PROGRAM AnalogConversion
VAR
	i					: INT := 1; //charger 1-6
	j					: INT := 1;  // section 1 - 4 
	k					: INT := 1;  // cap 1-10
	m					: INT := 1; //form cap 1-12
	n					: INT := 6;
	MaxTemp				: INT := 380;
	MinTemp				: INT := -70;
	
	MaxCurrent			: INT := 1000;
	MinCurrent			: INT := 0;
	
	MaxVolt				: INT := 105;
	//VoltMonAC1			: ARRAY[1..18] OF VoltMonAC_FB;
	//VoltMonAC2			: ARRAY[1..18] OF VoltMonAC_FB;
END_VAR

//MCP Charger 
//Analog Input
FOR i := 1 TO n BY 1 DO 
	//MCP_IO.Charger[i].voltageSP := (HMI_DB.TDKLoad[i].RequiredChargedV *1000);
	MCP_IO.Charger[i].voltageSP := (Setpoints.HPT5[i].RequiredChargedV);
END_FOR

//AI
FOR i := 1 TO n BY 1 DO
	//Temp
	MCP_IO.MagDriver[i].DumpResistorTemp_norm := Norm_x (raw_input := INT_TO_REAL (MCP_IO.MagDriver[i].DumpResistorTemp_raw),
														x_max := 32767,
														x_min := 6553); // temp sensor is 4-20mA
											
	MCP_IO.MagDriver[i].DumpResistorTemp := (MaxTemp - MinTemp) * ADC_10V( normal_input := MCP_IO.MagDriver[i].DumpResistorTemp_norm,
																			x_max := 10,
																			x_min := 2); // temp sensor is 2-10v
	//current																									
	MCP_IO.MagDriver[i].ShotCurrentFeedback_norm := Norm_x (raw_input := INT_TO_REAL (MCP_IO.MagDriver[i].ShotCurrentFeedback_raw),
														x_max := 32767,
														x_min := 0);
	
	MCP_IO.MagDriver[1].ShotCurrentFeedback := (MaxCurrent - MinCurrent) * ADC_10V( normal_input := MCP_IO.MagDriver[i].ShotCurrentFeedback_norm,
																							x_max := 10,
																							x_min := 0);

END_FOR;

//Analog Output
//voltageSP = Required Charge Voltage******************
//limit for charing the cap
//FOR i := 1 TO 8 BY 1 DO
FOR i := 1 TO n BY 1 DO	
	
	//set limits of charger voltage input 
	IF MCP_IO.Charger[i].voltageSP >= (MaxVolt) THEN
		MCP_IO.Charger[i].voltageSP := MaxVolt; //limit at 105V
	ELSIF MCP_IO.Charger[i].voltageSP <= 0 THEN
		MCP_IO.Charger[i].voltageSP := 0; //limit at 0V
	END_IF; 
		
	//prepare output signal for 50kV chargers.
	MCP_IO.Charger[i].voltageSP_norm := Norm_x (raw_input :=(MCP_IO.Charger[i].voltageSP), 
												x_max := MaxVolt,
												x_min := 0);	
												
	MCP_IO.Charger[i].voltageSP_raw := AQ (norm_input := MCP_IO.Charger[i].voltageSP_norm, 
												x_max := 20,
												x_min := 0);
																								
	//limite for output sigal (<= 10V)  this should not happen
	IF MCP_IO.Charger[i].voltageSP_raw >= (32767/2) THEN //32767/2
		MCP_IO.Charger[i].voltageSP_raw := (32767/2); 										
	END_IF;
	
END_FOR;

//no need for cap voltage feedback - the ultacap already scale those internally

//Cap voltage feedback
(*
//can also add a range of x samples for self calibrating **note: normalized range needs to be calibrated for each board
VoltMonitor_DB.VoltageReading_norm[0] := Norm_x (raw_input := INT_TO_REAL (VoltMonitor_DB.VoltageReading_raw[0]),
													x_max := 904, //10bit value - 1110001000 = 904deci
													x_min := 100); //100deci is the zero of range -1.61 to 12.01
LCP1_IO.Segment[1].Module[1].VoltageFeedback[1] := (12010 - 0) * ADC_10V(normal_input := VoltMonitor_DB.VoltageReading_norm[0],
																		x_max := 12.01,
																		x_min := 0); //use zero, it will cal for the -ve	

*)

(* // changed to a FB for norm and ADC
LCP1_IO.Segment[1].Module[1].VoltageFeedback_norm[1] := Norm_x (raw_input := INT_TO_REAL (LCP1_IO.Segment[1].Module[1].VoltageFeedback_raw[1]),
													x_max := 904, //10bit value - 1110001000 = 904deci
													x_min := 100); //100deci is the zero of range -1.61 to 12.01
LCP1_IO.Segment[1].Module[1].VoltageFeedback[1] := (12010 - 0) * ADC_10V(normal_input := LCP1_IO.Segment[1].Module[1].VoltageFeedback_norm[1],
																		x_max := 12.01,
																		x_min := 0); //use zero, it will cal for the -ve
*)

(*
// using FB instead.
VoltMonAC1[1](raw_input := DINT_TO_REAL(LCP1_IO.Segment[1].Module[1].VoltageFeedback_raw[1]),
				norm_x_max := 904, //individually calibrated, otherwise can do a for loop
				norm_x_min := 100, 
				RangUpp := 12.01, 
				RangLow := 0, 
				ADC_max := 12010, 
				ADC_min := 0, 
				voltage_reading => LCP1_IO.Segment[1].Module[1].VoltageFeedback[1]);
*)

					
//reset counter
//IF i > 8 THEN
IF i > n THEN
	i := 1;
END_IF;

IF j > 3 THEN 
	j := 1;
END_IF

IF k > 10 THEN 
	k := 1;
END_IF

IF m > 12 THEN 
	m := 1;
END_IF

END_PROGRAM

(* stored: Version 1.1.0.1, ProductVersion 3.1.4024.11
   POU AnalogConversion: Id {3b8eecca-a8e5-4cfd-bb8d-8865397a6f0b}, SpecialFunc None *)
